// Mitsubishi GX Works2 project: 응용   PLC: Q02/Q02H

PROGRAM MAIN
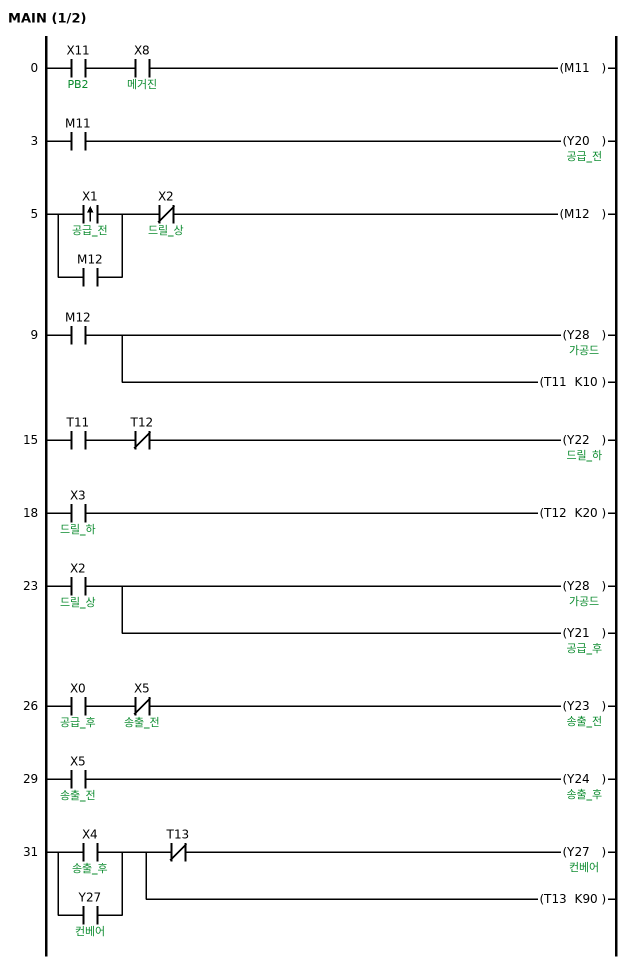
0     LD      X11  ; PB2
      AND     X8  ; 메거진
      OUT     M11
3     LD      M11
      OUT     Y20  ; 공급_전
5     LDP     X1  ; 공급_전
      OR      M12
      ANI     X2  ; 드릴_상
      OUT     M12
9     LD      M12
      OUT     Y28  ; 가공드
      OUT     T11 K10
15    LD      T11
      ANI     T12
      OUT     Y22  ; 드릴_하
18    LD      X3  ; 드릴_하
      OUT     T12 K20
23    LD      X2  ; 드릴_상
      OUT     Y28  ; 가공드
      OUT     Y21  ; 공급_후
26    LD      X0  ; 공급_후
      ANI     X5  ; 송출_전
      OUT     Y23  ; 송출_전
29    LD      X5  ; 송출_전
      OUT     Y24  ; 송출_후
31    LD      X4  ; 송출_후
      OR      Y27  ; 컨베어
      MPS
      ANI     T13
      OUT     Y27  ; 컨베어
      MPP
      OUT     T13 K90
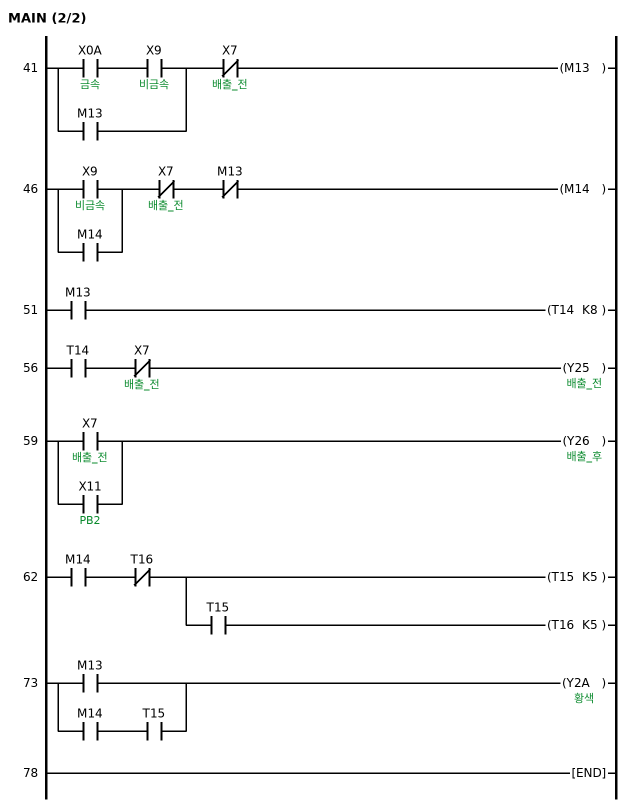
41    LD      X0A  ; 금속
      AND     X9  ; 비금속
      OR      M13
      ANI     X7  ; 배출_전
      OUT     M13
46    LD      X9  ; 비금속
      OR      M14
      ANI     X7  ; 배출_전
      ANI     M13
      OUT     M14
51    LD      M13
      OUT     T14 K8
56    LD      T14
      ANI     X7  ; 배출_전
      OUT     Y25  ; 배출_전
59    LD      X7  ; 배출_전
      OR      X11  ; PB2
      OUT     Y26  ; 배출_후
62    LD      M14
      ANI     T16
      OUT     T15 K5
      AND     T15
      OUT     T16 K5
73    LD      M13
      LD      M14
      AND     T15
      ORB
      OUT     Y2A  ; 황색
78    END
END_PROGRAM

// device comments not shown above
X6  ; 배출_후
X10  ; PB1
X12  ; PB3
Y29  ; 적색
Y2B  ; 녹색
